// TIA Portal V18 export
TYPE "PLCtoMES_AlarmMassage_ext"
// stored: IsFailsafeCompliant false
   STRUCT
      "MES.ErrorCode" : Int;   // 异常代码
      "MES.ErrorMsg" : String[60];   // 异常信息
   END_STRUCT;
END_TYPE
